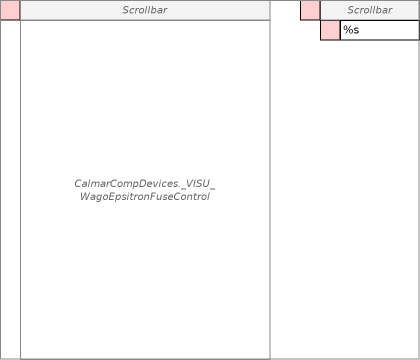
VISUALIZATION _VISU_PowerControl  // 420x360
VAR_IN_OUT
	mInst : FB_PowerControl;
END_VAR
    Frame (20,20 250x340)
        shows CalmarCompDevices._VISU_WagoEpsitronFuseControl(m_Inst_Fb := mInst.pEpsitronsInst[mInst.nEpsitronViewSel]^)
    RoundedRectangle (320,20 20x20), colour toggle: mInst.pFuseInputs[mInst.nFuseViewSel]^
    Scrollbar (320,0 100x20)
        p2245068023: mInst.nFuseInputsRegistered
        p1057716461: mInst.nFuseViewSel
    Rectangle (340,20 80x20), "%s", tooltip "%s", text variable: mInst.aFuseNames[mInst.nFuseViewSel]
        p4168582468: mInst.aFuseNames[mInst.nFuseViewSel]
    RoundedRectangle (300,0 20x20), tooltip "All Inputs ok", colour toggle: mInst.bO_AllFuseOk
    RoundedRectangle (0,0 20x20), tooltip "All Epsitron", colour toggle: mInst.bO_AllEpsitronOk
    Scrollbar (20,0 250x20)
        p2245068023: mInst.nEpsitronsRegistered
        p1057716461: mInst.nEpsitronViewSel
END_VISUALIZATION

(* stored: Version 1.1.0.1, ProductVersion 3.1.4024.11
   Visu _VISU_PowerControl: Id {25124c0c-27d8-416d-89f0-61b50931571a} *)
